// TIA Portal V19 export
DATA_BLOCK "CallEquipment_DB"   // DB96
AUTHOR : Siemens_FA_SUP
// stored: InstanceOfName Unit3.EM0.CallEquipment, InstanceOfType FB, Namespace Unit3.EM0
"Unit3.EM0.CallEquipment"
   // VAR_IN_OUT
   //    unitStatus : "LAF_typeUnitStatus";
   //    unitAlarmDB : "LAF_typeAlarms";
   //    emFeedback : "LUC_typeEmFeedback";
   // END_VAR
   // VAR
   //    statUnitStatus { ExternalWritable := 'False'} : "LAF_typeUnitStatus";
   //    instJob1 { ExternalWritable := 'False'} : "LAF_SelectJob";
   //    instSequence { ExternalWritable := 'False'} : "Unit3.EM0.Sequence";
   //    instManageBitAlarms { ExternalWritable := 'False'} : "LAF_ManageBitAlarms";
   // END_VAR
BEGIN
END_DATA_BLOCK
